Staubli VAL3: getPoint.pgx

public program getPoint(point& x_pPoint[], bool x_bCycle, num x_nIndex)
  local string l_sItem
  local num l_nSize
  local num i
  local num l_nPoint
begin
  // take
  if x_bCycle
    // in Cycle
    switch pt:tTraj[sItemCycle].tData[x_nIndex].nType
      case 0,2
        call getSizeItem(true,l_nSize)
        for i=0 to l_nSize-1
          // scan for the real point
          if pt:tTraj[sItemCycle].tData[i].nType==1
            l_nPoint=i
            i=l_nSize-1
          endIf
        endFor
        // give back
        x_pPoint=appro(pt:tTraj[sItemCycle].tData[l_nPoint].pPoint,pt:tTraj[sItemCycle].tData[x_nIndex].pPoint.trsf)
      break
      case 1
        // real point
        x_pPoint=pt:tTraj[sItemCycle].tData[x_nIndex].pPoint
      break
    endSwitch
  else
    // not in Cycle
    switch pEditPoint.tData[x_nIndex].nType
      case 0,2
        call getSizeItem(false,l_nSize)
        for i=0 to l_nSize-1
          // scan for the real point
          if pEditPoint.tData[i].nType==1
            l_nPoint=i
            i=l_nSize-1
          endIf
        endFor
        // give back
        x_pPoint=appro(pEditPoint.tData[l_nPoint].pPoint,pEditPoint.tData[x_nIndex].pPoint.trsf)
      break
      case 1
        // real point
        x_pPoint=pEditPoint.tData[x_nIndex].pPoint
      break
    endSwitch
  endIf
end
